gfCNCPoint3[29968] = {X 587.5870, Y 5.0000, Z -4.6667, A 0.000, B 0.000, C 0.000 }
gfCNCPoint3[29969] = {X 587.6872, Y 4.1099, Z -4.6667, A 0.000, B 0.000, C 0.000 }
gfCNCPoint3[29970] = {X 587.9831, Y 3.2645, Z -4.6667, A 0.000, B 0.000, C 0.000 }
gfCNCPoint3[29971] = {X 588.4596, Y 2.5060, Z -4.6667, A 0.000, B 0.000, C 0.000 }
gfCNCPoint3[29972] = {X 589.0930, Y 1.8727, Z -4.6667, A 0.000, B 0.000, C 0.000 }
gfCNCPoint3[29973] = {X 589.8514, Y 1.3961, Z -4.6667, A 0.000, B 0.000, C 0.000 }
gfCNCPoint3[29974] = {X 590.6969, Y 1.1003, Z -4.6667, A 0.000, B 0.000, C 0.000 }
gfCNCPoint3[29975] = {X 591.5870, Y 1.0000, Z -4.6667, A 0.000, B 0.000, C 0.000 }
gfCNCPoint3[29976] = {X 600.0000, Y 1.0000, Z -4.6667, A 0.000, B 0.000, C 0.000 }
gfCNCPoint3[29977] = {X 600.7927, Y 1.0793, Z -4.6667, A 0.000, B 0.000, C 0.000 }
gfCNCPoint3[29978] = {X 601.5540, Y 1.3142, Z -4.6667, A 0.000, B 0.000, C 0.000 }
gfCNCPoint3[29979] = {X 602.2537, Y 1.6953, Z -4.6667, A 0.000, B 0.000, C 0.000 }
gfCNCPoint3[29980] = {X 602.8639, Y 2.2075, Z -4.6667, A 0.000, B 0.000, C 0.000 }
gfCNCPoint3[29981] = {X 603.3605, Y 2.8305, Z -4.6667, A 0.000, B 0.000, C 0.000 }
gfCNCPoint3[29982] = {X 603.5431, Y 3.1435, Z -4.6667, A 0.000, B 0.000, C 0.000 }
gfCNCPoint3[29983] = {X 603.6966, Y 3.4718, Z -4.6667, A 0.000, B 0.000, C 0.000 }
gfCNCPoint3[29984] = {X 607.6966, Y 13.1476, Z -4.6667, A 0.000, B 0.000, C 0.000 }
gfCNCPoint3[29985] = {X 607.6966, Y 13.1476, Z -1.6667, A 0.000, B 0.000, C 0.000 }
gfCNCPoint3[29986] = {X 607.6966, Y 13.1476, Z 11.0000, A 0.000, B 0.000, C 0.000 }
gfCNCPoint3[29987] = {X 256.2445, Y 19.7811, Z 11.0000, A 0.000, B 0.000, C 0.000 }
gfCNCPoint3[29988] = {X 256.2445, Y 19.7811, Z -0.8333, A 0.000, B 0.000, C 0.000 }
gfCNCPoint3[29989] = {X 251.5292, Y 19.7811, Z -2.0968, A 0.000, B 0.000, C 0.000 }
gfCNCPoint3[29990] = {X 250.8345, Y 19.7919, Z -2.2830, A 0.000, B 0.000, C 0.000 }
gfCNCPoint3[29991] = {X 250.1812, Y 19.7933, Z -2.4580, A 0.000, B 0.000, C 0.000 }
gfCNCPoint3[29992] = {X 249.4952, Y 19.8918, Z -2.6437, A 0.000, B 0.000, C 0.000 }
gfCNCPoint3[29993] = {X 248.8453, Y 20.0800, Z -2.8250, A 0.000, B 0.000, C 0.000 }
gfCNCPoint3[29994] = {X 248.7083, Y 20.1113, Z -2.8627, A 0.000, B 0.000, C 0.000 }
gfCNCPoint3[29995] = {X 248.6543, Y 20.1620, Z -2.8825, A 0.000, B 0.000, C 0.000 }
gfCNCPoint3[29996] = {X 248.4753, Y 20.7649, Z -3.0510, A 0.000, B 0.000, C 0.000 }
gfCNCPoint3[29997] = {X 248.4452, Y 21.8674, Z -3.3466, A 0.000, B 0.000, C 0.000 }
gfCNCPoint3[29998] = {X 248.5584, Y 22.3425, Z -3.4774, A 0.000, B 0.000, C 0.000 }
gfCNCPoint3[29999] = {X 248.8739, Y 22.4373, Z -3.5657, A 0.000, B 0.000, C 0.000 }
gfCNCPoint3[30000] = {X 249.2022, Y 22.4644, Z -3.6540, A 0.000, B 0.000, C 0.000 }

ENDDAT
